// TIA Portal V19 export
VAR_GLOBAL   // PLC tag table "Default tag table"
   Stop_All AT %M0.0 : Bool;
END_VAR
